Fanuc KAREL source: KT00359.KL

PROGRAM KT00359
%NOLOCKGROUP
VAR
  P1: JOINTPOS
  P2: POSITION
  OUT: BOOLEAN
BEGIN
  OUT = P1 < P2
END KT00359
